// TIA Portal project "TermikSantralBuharKazaniKontrolUygulamasi" (V17)

(* hardware
DEVICE "S7-1500/ET200MP station_1"  S7-1500 station
   slot 0: "Rail_0"  Rack  6ES7 590-1***0-0AA0
   slot 1: "PLC_1"  CPU 1515F-2 PN  6ES7 515-2FM02-0AB0  V2.9
      slot 3: "CPU display_1"  6ES7591-1BA00-0AA0
      slot 32768: "PROFINET interface_1"  X1
         slot 32769: "Port_1"  X1 P1
         slot 32770: "Port_2"  X1 P2
      slot 33024: "PROFINET interface_2"  X2
         slot 33025: "Port_1"  X2 P1
      slot 34817: "Virtual CP interface port_1"  Virtual CP interface port  Virtual CP interface port
*)

// ===== PLC "PLC_1"  CPU 1515F-2 PN =====

VAR_GLOBAL   // PLC tag table "Default tag table"
   "IŞIKLI UYARI" AT %Q124.0 : Bool;
   "ALARM SİNYALİ" AT %I124.0 : Bool;
   "Tag_1" AT %C0 : Counter;
   "Tag_2" AT %T0 : Timer;
   "Tag_3" AT %T1 : Timer;
END_VAR

DATA_BLOCK "Main_Safety_RTG1_DB"   // DB1, F_DB
{ S7_Optimized_Access := 'TRUE' }
NAME : FUSI
VERSION : 0.1
// stored: InstanceOfName Main_Safety_RTG1
"Main_Safety_RTG1"
BEGIN
END_DATA_BLOCK

FUNCTION_BLOCK "Main_Safety_RTG1"   // FB1, F_FBD
{ S7_Optimized_Access := 'TRUE' }
BEGIN
END_FUNCTION_BLOCK

ORGANIZATION_BLOCK "Main"   // OB1, LAD, ProgramCycle
TITLE = "Main Program Sweep (Cycle)"
{ S7_Optimized_Access := 'TRUE' }
VERSION : 0.1
   VAR_INPUT
      Initial_Call : Bool;   // Initial call of this OB
      Remanence : Bool;   // =True, if remanent data are available
   END_VAR
BEGIN

REGION Network 1
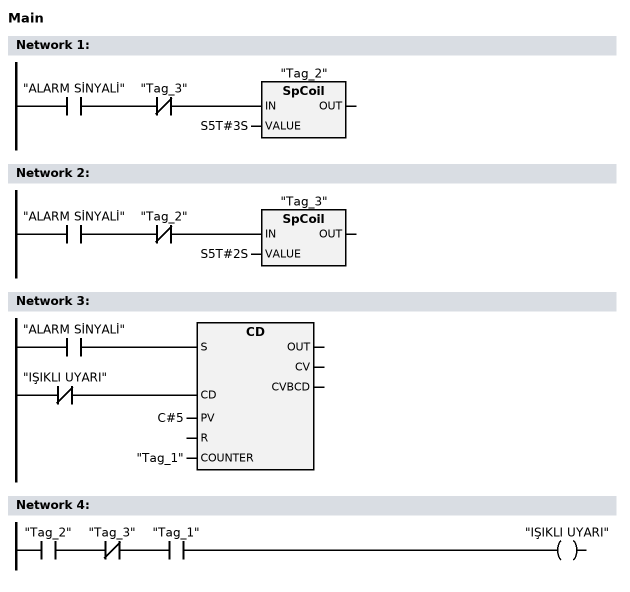
   // no SCL statement known for SpCoil: written as a call
   SpCoil(in := "ALARM SİNYALİ" AND NOT "Tag_3", value := S5T#3S, operand := "Tag_2");
END_REGION

REGION Network 2
   // no SCL statement known for SpCoil: written as a call
   SpCoil(in := "ALARM SİNYALİ" AND NOT "Tag_2", value := S5T#2S, operand := "Tag_3");
END_REGION

REGION Network 3
   // no SCL statement known for Cd: written as a call
   Cd(cd := NOT "IŞIKLI UYARI", s := "ALARM SİNYALİ", pv := C#5, "counter" := "Tag_1");
END_REGION

REGION Network 4
   RUNG wire#powerrail
      Contact( "Tag_2" )
      I_Contact( "Tag_3" )
      Contact( "Tag_1" )
      Coil( "IŞIKLI UYARI" )
   END_RUNG
   // the same network as SCL:
   "IŞIKLI UYARI" := "Tag_2" AND NOT "Tag_3" AND "Tag_1";
END_REGION
END_ORGANIZATION_BLOCK